PROGRAM MAIN
VAR
END_VAR

(* Update physical IO signals *)
F_UpdateIO();

(* Update transport tubes *)
GVL_TransportTubes.fbLS1(
	i_stConfig := GVL_TransportTubes.stLS1, 
	i_bLaserExtIntl := TRUE
);

GVL_TransportTubes.fbLS5(
	i_stConfig := GVL_TransportTubes.stLS5, 
	i_bLaserExtIntl := TRUE
);

GVL_TransportTubes.fbLS8(
	i_stConfig := GVL_TransportTubes.stLS8, 
	i_bLaserExtIntl := TRUE
);

GVL_TransportTubes.fbLD2(
	i_stConfig := GVL_TransportTubes.stLD2,
	i_bLaserExtIntl := TRUE
);

GVL_TransportTubes.fbLD4(
	i_stConfig := GVL_TransportTubes.stLD4,
	i_bLaserExtIntl := TRUE
);

GVL_TransportTubes.fbLD6(
	i_stConfig := GVL_TransportTubes.stLD6,
	i_bLaserExtIntl := TRUE
);

GVL_TransportTubes.fbLD14(
	i_stConfig := GVL_TransportTubes.stLD14,
	i_bLaserExtIntl := TRUE
);

GVL_TransportTubes.fbLD10(
	i_stConfig := GVL_TransportTubes.stLD10,
	i_bLaserExtIntl := TRUE
);

GVL_TransportTubes.fbLD9(
	i_stConfig := GVL_TransportTubes.stLD9,
	i_bLaserExtIntl := TRUE
);

GVL_TransportTubes.fbLD8(
	i_stConfig := GVL_TransportTubes.stLD8,
	i_bLaserExtIntl := TRUE
);

END_PROGRAM

(* stored: Version 1.1.0.1, ProductVersion 3.1.4022.18
   POU MAIN: Id {e39c3acf-17bf-44fe-a884-c77329dee9c5}, SpecialFunc None *)
